FUNCTION_BLOCK QXP (* Composite FB for boolean output data *)
  (* Standard: 61499-2 *)
  (* Version 1.0, 2024-04-24, franz *)
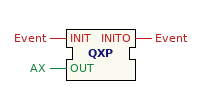
  EVENT_INPUT
    INIT; (* Initialization Request *)
  END_EVENT
  EVENT_OUTPUT
    INITO; (* Initialization Confirm *)
  END_EVENT
  SOCKETS
    OUT : AX;
  END_SOCKETS
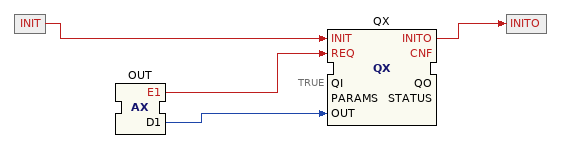
  FBS
    QX : QX(QI := TRUE);
  END_FBS
  EVENT_CONNECTIONS
    INIT TO QX.INIT;
    QX.INITO TO INITO;
    OUT.E1 TO QX.REQ;
  END_CONNECTIONS
  DATA_CONNECTIONS
    OUT.D1 TO QX.OUT;
  END_CONNECTIONS
END_FUNCTION_BLOCK
